(* IEC 61131-3 sources: Industry-PLC-LLM/data/PLCBEAD_repo/PLCBEAD_PLCEmbed-main/PLC-BEAD/Source/GEB/ARRAY_SPR, 1 file *)

(* ---- ARRAY_SPR.ST ---- *)
TYPE
	oscat_PT_ARRAY: ARRAY [1..100] OF REAL;
END_TYPE

FUNCTION_BLOCK ARRAY_SPR_Block
	VAR_IN_OUT
		PT :	oscat_PT_ARRAY;
	END_VAR

	VAR_INPUT
		SIZE :	UINT;
	END_VAR

	VAR_OUTPUT
		ARRAY_SPR :	REAL;
	END_VAR

	VAR
		i :	INT;
		STOP :	INT;
		array_max :	REAL;
		ARRAY_MIN :	REAL;
	END_VAR

	STOP :=LIMIT_INT(1,UINT_TO_INT(SIZE),1000);

	ARRAY_MIN := PT[1];
	array_max := PT[1];
	FOR i := 2 TO STOP DO
		IF PT[i] > array_max THEN array_max := PT[i];
		ELSIF PT[i] < ARRAY_MIN THEN ARRAY_MIN := PT[i];
		END_IF;
	END_FOR;
	ARRAY_SPR := array_max - ARRAY_MIN;
END_FUNCTION_BLOCK

PROGRAM program0
  VAR
    LocalVar0 : oscat_PT_ARRAY;
    LocalVaR1  : UINT;
	LocalOUT  : REAL;
	func_block : ARRAY_SPR_Block;
  END_VAR
	func_block(PT := LocalVar0,SIZE := LocalVaR1 );
	LocalOUT := func_block.ARRAY_SPR;

END_PROGRAM
